{attribute addProperty BoxType "EK1122-0000-0018"}
{attribute addProperty Id "Beckhoff_EJ6xxxsub_EK1100EK1100_179A0949162"}
{attribute addProperty CRC "813144453"}
{attribute addProperty SizeInBites "16"}
{attribute addProperty SizeInBytes "2"}
TYPE Beckhoff_EJ6xxxEK1122_30779985 EXTENDS EK1122_179A0949 :
STRUCT
	{attribute addProperty Name "Beckhoff_EJ6xxxsub_EK1100"}
	Beckhoff_EJ6xxxsub_EK1100 : EK1100_179A0949;
END_STRUCT
END_TYPE

(* stored: Version 1.2.0.0, ProductVersion 3.1.4024.9
   DUT Beckhoff_EJ6xxxEK1122_30779985: Id {a1ca1ec7-c0bf-4216-bfb8-1d3cad0f5894} *)
